{attribute 'qualified_only'}
VAR_GLOBAL
//Input to PLC from process
	ixAGVStrobe		AT %I*:	BOOL;	(* AGV strobe signal *)
	iiAtPos			AT %I*:	INT;	(* Actual position of AGV *)
	
//Output from PLC to process
	qxPLCStrobe		AT %Q*:	BOOL;	(* PLC strobe signal *)
	qiGotoPos		AT %Q*:	INT;	(* Target position for AGV *)
// ADD THESE for R1 route control
    xStart         : BOOL := FALSE;
    iOrder         : INT  := 0;
    xStop          : BOOL := FALSE;
	OrderRobot_0   : OrderRobot;
// R2 data transmission
    sLocation      : STRING := '';
    iBattery       : INT    := 75;
    xSendNow       : BOOL   := FALSE;
END_VAR

(* stored: Version 1.1.0.1
   GVL GVL: Id {816111f0-16ef-4f4d-a70e-f3df38e5b1aa} *)
